// TwinCAT 3 PLC project CL_TelegramTxtLogLibrary
// Title: CL_TelegramTxtLogLibrary
// Company: CleanGreens SA
// Author: Massimo Lucano
// ProjectVersion: 2.2
// Description: Telegram API implementation, TextLOg implementation, Link between CL_DefectManager and Telegram and TextLog
// ProgramVersion: 3.1.4024.0
// libraries:
//   CL_DefectManager, * (CleanGreens SA)
//   CL_ErrorsDatabase, * (CleanGreens SA)
//   CL_CleanGreensObjectsLibrary, * (CleanGreens SA)
//   Tc2_Standard, * (Beckhoff Automation GmbH)
//   Tc2_System, * (Beckhoff Automation GmbH)
//   Tc2_Utilities, * (Beckhoff Automation GmbH)
//   Tc3_IotBase, * (Beckhoff Automation GmbH)
//   Tc3_IotCommunicator, * (Beckhoff Automation GmbH)
//   Tc3_JsonXml, * (Beckhoff Automation GmbH)
//   Tc3_Module, * (Beckhoff Automation GmbH)
// project tree:
//   DUTs/ enBOT_API.TcTLEO, E_MsgType.TcDUT, ST_getMe.TcDUT, ST_TelegramInit.TcDUT
//   / PlcTask.TcTTO
//   POUs/ CL_LinkDefectMgrToTelegramAndLog.TcPOU, CL_TelegramBOT.TcPOU, CL_TextLog.TcPOU
// real-time tasks:
//   TASK PlcTask: cycle T#10ms, priority 20, ADS port 350

CONFIGURATION CL_TelegramTxtLogLibrary
    RESOURCE PLC ON TwinCAT3
        TASK PlcTask(INTERVAL := T#10ms, PRIORITY := 20);
        PROGRAM Main WITH PlcTask : Main;
    END_RESOURCE
END_CONFIGURATION

// ---- DUTs/enBOT_API.TcTLEO
TYPE enBOT_API :
(
	none := 0, getMe := 1, sendMsg := 2, getUpdates := 3
);
END_TYPE

// ---- DUTs/E_MsgType.TcDUT
{attribute 'qualified_only'}
{attribute 'strict'}
TYPE E_MsgType :
(
	Alarm := 0,
  Info,
  Register
);
END_TYPE

// ---- DUTs/ST_getMe.TcDUT
TYPE ST_getMe :
STRUCT
	id 						              : ULINT;
	first_name				          : T_MaxString;//BOT name
	username				            : T_MaxString;//owner name
  is_bot					            : BOOL;
	can_join_groups			        : BOOL;
	can_read_all_group_messages : BOOL;
	supports_inline_queries	    : BOOL;
END_STRUCT
END_TYPE

// ---- DUTs/ST_TelegramInit.TcDUT
TYPE ST_TelegramInit :
STRUCT
  sBOTKey   		  : STRING(64);//BOT key to exchange operator messages
	sDebugID   		  : STRING(32);//chat group ID to send debug messages Info et Verbose
	sAlarmID   		  : STRING(32);//chat group ID to send Critical,Error,Warning alarms
	sBOTname  		  : STRING(40);
	sBOTusername  	: STRING(40);
END_STRUCT
END_TYPE

// ---- POUs/CL_LinkDefectMgrToTelegramAndLog.TcPOU
{attribute 'enable_dynamic_creation'}
FUNCTION_BLOCK CL_LinkDefectMgrToTelegramAndLog EXTENDS CL_MasterRootClass
VAR
  bInit                   : BOOL := FALSE;
	_DefectMngr             : REFERENCE TO CL_DefectManager;
  _TelegramBOT            : REFERENCE TO CL_TelegramBOT;
  _TxtLog                 : REFERENCE TO CL_TextLog;
  _ActTime                :	REFERENCE TO CL_ActTimeDate;
  
  indListAll 					    : UINT := 1;
  indListAct  				    : UINT := 1;

  _stConfigMsgBuild       : ST_ConfigMsgBuild;
  _stShow                 : ST_ShowMsgFields;
  
  _bShowRegisterMsg       : BOOL := FALSE;
  _bAllDefectsRegistered  : BOOL := FALSE;
	
	sTelegramMsg_P	        : POINTER TO T_StringBuffer;//used to generate very long Telegram messages limited to 3500 chars
	sTextOut_P              : POINTER TO T_StringBuffer;//used to generate short ADS console messages limited to 255 chars
  
	pDf			      		      : POINTER TO CL_Defect;
	iDf		        		      : ITF_Defect;
END_VAR

IF bInit THEN
  this^.Run(); 
END_IF

METHOD PRIVATE AddDateTime
VAR_IN_OUT
	sMsgTimeCreation	: T_MaxString;
END_VAR
VAR
  sDatetime         : T_MaxString;
END_VAR
(*
sBOTMsgTimeCreation^ := DT_TO_STRING(_objActTime_R.GetDateTime);
sBOTMsgTimeCreation^ := REPLACE(sBOTMsgTimeCreation^,' ',1,3);
sBOTMsgTimeCreation^ := CONCAT(' ',sBOTMsgTimeCreation^);
//sBOTMsgTimeCreation^ := CONCAT(sBOTMsgTimeCreation^,'%0A');
sBOTMsgTimeCreation^ := CONCAT(sBOTMsgTimeCreation^,'  ');
*)

(*
sMsgTimeCreation := concat(sMsgTimeCreation,_ActTime.GetStrDateTime());//2024-10-15-23:16:25
sMsgTimeCreation := REPLACE(sMsgTimeCreation,' ',1,11);
sMsgTimeCreation := CONCAT('Date: ', sMsgTimeCreation);
sMsgTimeCreation := CONCAT(sMsgTimeCreation,'  ');
*)

sMsgTimeCreation := CONCAT(sMsgTimeCreation,'  Date: ');
sDatetime := _ActTime.GetStrDateTime();//2024-10-15-23:16:25
sDatetime := REPLACE(sDatetime,' ',1,11);
sMsgTimeCreation := CONCAT(sMsgTimeCreation,sDatetime);
END_METHOD

PROPERTY PUBLIC AllDefectsRegistered : BOOL
GET
AllDefectsRegistered := _bAllDefectsRegistered;
END_GET
SET
_bAllDefectsRegistered := AllDefectsRegistered;
END_SET
END_PROPERTY

METHOD PRIVATE BuildMsg : BOOL
VAR_INPUT
  MsgType       : E_MsgType;
END_VAR
VAR
  sStartMsg     : T_MAXSTRING;
  
END_VAR
//%0A telegram new line
CASE MsgType OF
  E_MsgType.Alarm:
    sStartMsg := _stConfigMsgBuild.AlarmMsg.sStartMsg;
    _stShow := _stConfigMsgBuild.AlarmMsg;
  E_MsgType.Info:
    sStartMsg := _stConfigMsgBuild.InfoMsg.sStartMsg;
    _stShow := _stConfigMsgBuild.InfoMsg;
  E_MsgType.Register:
    sStartMsg := _stConfigMsgBuild.RegisterMsg.sStartMsg;
    _stShow := _stConfigMsgBuild.RegisterMsg;
END_CASE   
sTelegramMsg_P^ := '';
sTextOut_P^ := '';

BuildMsg := pDf^.BuildStringMsg(sMsgOut_P := sTelegramMsg_P, sTextOut_P := sTextOut_P, stShow := _stShow);
                                      
IF _stShow.bDateTime THEN 
  AddDateTime(sStartMsg);
END_IF  

IF _stShow.bTelegram THEN
  CONCAT2(ADR(sStartMsg),sTelegramMsg_P,sTelegramMsg_P,SIZEOF(sTelegramMsg_P^));
END_IF

IF _stShow.bTxtLog THEN
  CONCAT2(ADR(sStartMsg),sTextOut_P,sTextOut_P,SIZEOF(sTextOut_P^));
END_IF
END_METHOD

METHOD PUBLIC Init : BOOL
VAR_INPUT
  stIrrLine        : ST_LineReference;
  DefectMngr       : REFERENCE TO CL_DefectManager;
  TelegramBOT      : REFERENCE TO CL_TelegramBOT;
  TxtLog           : REFERENCE TO CL_TextLog;
  ActTime          : REFERENCE TO CL_ActTimeDate;
  stConfigMsg      : ST_ConfigMsgBuild;
END_VAR
VAR
  bufferSize       : UDINT;
END_VAR
bInit := Init := FALSE;
IF __ISVALIDREF(DefectMngr) AND __ISVALIDREF(TelegramBOT) AND __ISVALIDREF(TxtLog) and __IsValidRef(ActTime) THEN 
	_DefectMngr REF= DefectMngr;
  _TelegramBOT REF= TelegramBOT;
  _TxtLog REF= TxtLog;
  _ActTime REF= ActTime;
  
  MRCLineRef := stIrrLine;

  indListAll := indListAct := 1;

	_stConfigMsgBuild := stConfigMsg;
  _bShowRegisterMsg := _stConfigMsgBuild.bShowRegisterMsg;
  
  bufferSize := SIZEOF(T_StringBuffer)+4;
  sTelegramMsg_P := __NEW(BYTE, bufferSize);
  sTextOut_P := __NEW(BYTE, bufferSize);

  bInit := Init := sTelegramMsg_P <> 0 AND sTextOut_P <> 0;
END_IF
END_METHOD

PROPERTY PUBLIC RegisterAllMsgSent : BOOL
GET
RegisterAllMsgSent := not _bShowRegisterMsg;
END_GET
END_PROPERTY

METHOD PUBLIC Release : BOOL
bInit := FALSE;
IF sTelegramMsg_P <> 0  THEN 
  __DELETE(sTelegramMsg_P);
END_IF

IF sTextOut_P <> 0  THEN 
  __DELETE(sTelegramMsg_P);
END_IF

Release := sTelegramMsg_P = 0 AND sTextOut_P = 0;
END_METHOD

METHOD PRIVATE Run
VAR
  bDefectToSend	: BOOL;
END_VAR
IF NOT _TelegramBOT.IsBusy AND NOT _TxtLog.IsBusy THEN  
  
  IF _bShowRegisterMsg  THEN
    pDf := _DefectMngr.ListAll(indListAll,0);
    IF pDf <> 0 THEN
      iDf := pDf^;
      IF __QUERYPOINTER(iDf, pDf) THEN // Ctrl if address has the good interface (ITF_Default)
        RunRegister();
      END_IF//__QUERYPOINTER
    END_IF//_DefectMngr.List(indDfList,0) <> 0 
    //Telegram and TextLog not Busy --> increment at each cycle the Defect index
    indListAll := indListAll + 1;
    IF (indListAll > _DefectMngr.nMaxDefects) THEN //all Defect Register Messages sent
      indListAll := 1;
      //after first pass all register messages are sent, do not send anymore
      //the object can send starting from now Alarm and Info messages
      _bShowRegisterMsg := FALSE;
    END_IF 
  END_IF//_bShowRegisterMsg
  
  IF NOT _bShowRegisterMsg  THEN
    pDf := _DefectMngr.ListCurrent(indListAct);
    IF pDf <> 0 THEN
      iDf := pDf^;
      IF __QUERYPOINTER(iDf, pDf) THEN // Ctrl if address has the good interface (ITF_Default)
        IF pDf^.DefectToSend THEN 
          RunAlarm();
          RunInfo();
        END_IF
      END_IF//__QUERYPOINTER
    END_IF//_DefectMngr.ListCurrent(indDfList,0) <> 0 
    indListAct := indListAct + 1;
    IF (indListAct > _DefectMngr.nMaxDefectsView) THEN
      indListAct := 1;
    END_IF 
  END_IF//not _bShowRegisterMsg
ELSE
  //ADSLOGSTR(ADSLOG_MSGTYPE_LOG, 'Telegram busy','');//only for debug
  IF _TelegramBOT.IsError THEN 
    ADSLOGSTR(ADSLOG_MSGTYPE_LOG, 'Telegram error: Telegram server answer with HTTP error','');
  END_IF
END_IF//TelegramBOT and TextLog both are not busy
END_METHOD

METHOD PRIVATE Run_old
VAR
  bDefectToSend	: BOOL;
END_VAR
(*
IF NOT _TelegramBOT.IsBusy AND NOT _TxtLog.IsBusy THEN  
  
	IF _DefectMngr.List(indDfList,0) <> 0 THEN
		iDf := _DefectMngr.List(indDfList,0)^;
		IF __QUERYPOINTER(iDf, pDf) THEN // Ctrl if address has the good interface (ITF_Default)
      pDf := _DefectMngr.List(indDfList,0);  
      IF _bShowRegisterMsg then
        RunRegister();
        IF (indDfList > _DefectMngr.nMaxDefects) THEN //all Defect Register Messages sent
          _bShowRegisterMsg := false;//Register all defects done; the object can send starting from now Alarm and Info messages
				END_IF
			ELSE
        //condition OR pDf^.State = E_DefectState.OffAndNotAck added MPL date 16-11-2024
        bDefectToSend := pDf^.State = E_DefectState.Active OR pDf^.State = E_DefectState.ActiveAndAck OR pDf^.State = E_DefectState.OffAndNotAck;
        IF bDefectToSend THEN 
          RunAlarm();        
          RunInfo();
        END_IF
      END_IF
    END_IF//__QUERYPOINTER
  END_IF//_DefectMngr.List(indDfList,0) <> 0 

  //Telegram and TextLog not Busy --> increment at each cycle the Defect index
  indDfList := indDfList + 1;
  IF (indDfList > _DefectMngr.nMaxDefects) THEN	// Constant not accessible defect manager, or yes. Actually yes, but access through GVL not suitable!	
    indDfList := 1;
    _bShowRegisterMsg := false;//after first pass all register messages are sent, do not send anymore
  END_IF 
END_IF//TelegramBOT and TextLog both are not busy
*)
END_METHOD

METHOD PRIVATE RunAlarm
VAR_INPUT
END_VAR
//TcEventSeverity : (Verbose:=0, Info:=1, Warning:=2, Error:=3, Critical:=4);
IF pDf^.CanSendAlarmMsg AND (pDf^.Severity > TcEventSeverity.Info) THEN //Telegram msg not yet sent   
  //Critical, Error and Warning Defect are sent to Alarm group
  IF BuildMsg(E_MsgType.Alarm) THEN
    IF _stShow.bTxtLog THEN 
      _TxtLog.RequWriteMsg(sTextOut_P);
    END_IF
    IF _stShow.bTelegram THEN
      _TelegramBOT.RequSendMsgToAlarm(sTelegramMsg_P);
    END_IF
  END_IF					
END_IF//pDf^.Severity... and pDf^.CanSendTelegramAlarmMsg
END_METHOD

METHOD PRIVATE RunInfo
VAR_INPUT
END_VAR
//TcEventSeverity : (Verbose:=0, Info:=1, Warning:=2, Error:=3, Critical:=4);
//sendMsgToAlarm and sendMsgToInfo cannot be executed together; sendMsgToInfo can be requested only once AlarmMsgAlreadySent is true and TelegramBOT is again not busy
//IF (pDf^.CanSendInfoMsg AND (pDf^.Severity <= TcEventSeverity.Info)) OR (pDf^.CanSendInfoMsg AND (pDf^.Severity > TcEventSeverity.Info) AND pDf^.AlarmMsgAlreadySent) THEN
IF (pDf^.CanSendInfoMsg AND (pDf^.Severity <= TcEventSeverity.Info)) THEN
  //Verbose and Info Defect are sent only to InfoDebug group
  IF BuildMsg(E_MsgType.Info) THEN
    IF _stShow.bTelegram THEN
      _TelegramBOT.RequSendMsgToInfo(sTelegramMsg_P);
    END_IF
    IF _stShow.bTxtLog THEN 
      _TxtLog.RequWriteMsg(sTextOut_P);
    END_IF
  END_IF
END_IF//pDf^.Severity... and pDf^.CanSendTelegramAlarmMsg
END_METHOD

METHOD PRIVATE RunRegister
IF pDf^.CanSendRegisterMsg AND _bShowRegisterMsg THEN //all Defect registered are sent
  IF BuildMsg(E_MsgType.Register) THEN
   IF _stShow.bTxtLog THEN 
    _TxtLog.RequWriteMsg(sTextOut_P);
   END_IF
   IF _stShow.bTelegram THEN
    _TelegramBOT.RequSendMsgToInfo(sTelegramMsg_P);
   END_IF
  END_IF
END_IF
END_METHOD

METHOD PRIVATE TelegramMsgFilter : BOOL
VAR_INPUT
	sDatabaseMsg	:	T_MaxString;
END_VAR
VAR_OUTPUT
	sTelegramMsg	:	T_MaxString;
END_VAR
VAR
	sTelegramTmp	:	T_MaxString;
	i:	INT;
	iSafe:	INT;
	iLengthStr:	INT	:= 0;
	iNonAsciiPos:	INT;
	iNumAsciiChar:	UDINT;

END_VAR

VAR CONSTANT
		// Language tables - hardcoded here since part of the algorithm, and meaningless to keep them outside.
	sASCIIcompatCharFR_AR : ARRAY [1..2,1..28] OF STRING := ['à','â','é','è','ê','ë','î','ï','ô','ù','û','ü','ÿ','ç',
																															'À','Â','É','È','Ê','Ë','Î','Ï','Ô','Ù','Û','Ü','Ÿ','Ç',
																															2('a'),4('e'),2('i'),'o',3('u'),'y','c',
																															2('A'),4('E'),2('I'),'O',3('U'),'Y','C'];
	sASCIIcompatCharDE_AR :	ARRAY [1..2,1..7] OF STRING  := ['Ä','ä','Ö','ö','Ü','ü','ß',
																															'Ae','ae','Oe','oe','Ue','ue','ss'];
END_VAR

sTelegramTmp := sDatabaseMsg;
IF NOT F_StringIsASCII(pSTRING := ADR(sTelegramTmp), nLen => iNumAsciiChar) THEN
	iLengthStr := LEN(sTelegramTmp);
//	IF C.sLangErrors = 'fr' THEN
	IF  _DefectMngr.ErrorDB.sMsgLang = 'fr' THEN
			FOR i:=1 TO 28 BY 1 DO
				iSafe := 0;
				REPEAT
					iNonAsciiPos := FIND(sTelegramTmp,sASCIIcompatCharFR_AR[1,i]);	// Table to store inside the object, as never used elsewhere and fixed sized.
					IF iNonAsciiPos <> 0 THEN
						sTelegramTmp := REPLACE(sTelegramTmp,sASCIIcompatCharFR_AR[2,i],1,iNonAsciiPos);
					END_IF
					iSafe := iSafe + 1;
				UNTIL iNonAsciiPos = 0 OR iSafe > iLengthStr
				END_REPEAT;	
			END_FOR
//	ELSIF C.sLangErrors = 'de' THEN
	ELSIF  _DefectMngr.ErrorDB.sMsgLang = 'de' THEN
		FOR i:=1 TO 7 BY 1 DO
		iSafe := 0;
			REPEAT
				FIND(sTelegramTmp,sASCIIcompatCharDE_AR[1,i]);
				IF iNonAsciiPos <> 0 THEN
					REPLACE(sTelegramTmp,sASCIIcompatCharDE_AR[2,i],1,iNonAsciiPos); // Caution, the length of the string is increasing
				END_IF
			iSafe := iSafe + 1;
			UNTIL iNonAsciiPos = 0 OR iSafe > 2*iLengthStr
			END_REPEAT
		END_FOR
	END_IF
END_IF
sTelegramMsg := sTelegramTmp;

//only to reproduce the bug without filtering
//sTelegramMsg := sDatabaseMsg;
END_METHOD

END_FUNCTION_BLOCK

// ---- POUs/CL_TelegramBOT.TcPOU
{attribute 'enable_dynamic_creation'}
FUNCTION_BLOCK CL_TelegramBOT EXTENDS CL_MasterRootClass
VAR CONSTANT //constant configuration parameters fro FB_IotHttpClient configuration
	sHostNameC 					: T_MaxString:='api.telegram.org';
	nHostPortC  				: UINT := 443; //https port
	bKeepAliveC 				: BOOL := FALSE;
	bNoServerCertCheckC : BOOL := TRUE;
	tConnectionTimeoutC : TIME := T#10S;
END_VAR
VAR
	boBOT_MSGOk 				: BOOL := FALSE;
		
	sBOTKey 						: T_MaxString;// BOT key to exchange operator messages
	sDebugID 						: STRING(64);//32
	sAlarmID 						: STRING(64);//32
	sBOTname 						: STRING(64);//40
	sBOTusername 				: STRING(64);//40
	
	bInit		            : BOOL := FALSE;
 	
	fbHttpClientTelegram: FB_IotHttpClient;//HTTP client communication
	fbBOTRequest   			: FB_IotHttpRequest;
	
	sBOTMsgBuffer_P			: POINTER TO T_StringBuffer;//STRING(2000);//string buffer
	sBOT_APIMethod_P 		: POINTER TO T_StringBuffer;//STRING(3500);//used in HTTPGetTelegram
	sBOTReturnContent_P : POINTER TO T_StringBuffer;//STRING(2000);//used in HTTPGetTelegram
  
	RisingEdge          : R_TRIG;
	HTTPGetTelegramStm  : BYTE := 0;
  nBOTReqCnt          : UDINT := 0;    
  nBOTContentCnt      : UDINT := 0;
    
  nErrCount           : UDINT;
	bBOTSend						: BOOL;
	bBOTHTTPError			  : BOOL := FALSE;
	bBOTBusy            : BOOL := FALSE; 
	
	//used in
	bJSONReturnExec			: BOOL := FALSE;
	JSONReturnStm				: enBOT_API := enBOT_API.none;
	nJSONResCnt         : UDINT := 0;
	
	//returned values from getMe
	stJsonGetMe					: ST_getMe;
	bJsonGetMe					: BOOL;
	bBOTCorret					: BOOL  := TRUE; //the BOT is correctly identified after the initial getMe Api call 
END_VAR
{attribute 'TcEncoding':='UTF-8'}

//IMPORTANT ATTENTION: forbidden words for Telegram messages otherwise FB_IotHttpRequest FAILS!! Forbidden words: HandlingLine HMI
IF bInit THEN
	IF fbHttpClientTelegram.bConfigured AND bBOTCorret THEN
		fbHttpClientTelegram.Execute();
		HTTPGetTelegramExec();
		JSONBOTReturnExec();
	END_IF
END_IF

METHOD PRIVATE HTTPGetTelegramExec
VAR
   nBOTReturnContentSize 		: UDINT;
	 HTTPStatusCodeFromServer	: UINT;
END_VAR
IF (bBOTSend) THEN
	RisingEdge(CLK:= TRUE );
	CASE HTTPGetTelegramStm OF
		0: IF RisingEdge.Q THEN 
				IF fbBOTRequest.SendRequest(sUri:=sBOT_APIMethod_P^, fbClient:=fbHttpClientTelegram, eRequestType:=ETcIotHttpRequestType.HTTP_Get, 0, 0, 0) THEN                
					HTTPGetTelegramStm:= 1;
					nBOTReqCnt:= nBOTReqCnt+1;
					bBOTBusy:= TRUE;
					bBOTHTTPError:= FALSE;
				END_IF                    
    	END_IF
		1: IF NOT fbBOTRequest.bBusy THEN
        bBOTHTTPError:= TRUE;
        IF NOT fbBOTRequest.bError THEN  
          bBOTHTTPError:= NOT fbBOTRequest.GetContent(pContent:= sBOTReturnContent_P,
					nContentSize:= nBOTReturnContentSize:= SIZEOF(T_StringBuffer),
					bSetNullTermination:= TRUE);
					IF JSONReturnStm = enBOT_API.getUpdates THEN
						bBOTHTTPError := FALSE;
						//the JSON answer from getUpdates methos could be very large; in this case a truncated answer will be stored in sBOTReturnContent
						//fbBOTRequest.GetContent will return an error -> in this case the error is always cleared
					END_IF
					bBOTSend := FALSE; //do not execute any longer HTTPGetTelegramExec
					//bBOTError:= FALSE -> ok sBOTReturnContent returned good value
					HTTPStatusCodeFromServer := fbBOTRequest.nStatusCode;
					IF NOT bBOTHTTPError AND HTTPStatusCodeFromServer >= 200 AND HTTPStatusCodeFromServer < 300 THEN
						bJSONReturnExec := TRUE;
						nBOTContentCnt:= nBOTContentCnt+1;
					ELSE
						bBOTHTTPError := TRUE;//server answer with HTTP error
            //ADSLOGSTR(ADSLOG_MSGTYPE_LOG, 'Telegram error: Telegram server answer with HTTP error','');//only debug
					END_IF
        END_IF
				RisingEdge(CLK:= FALSE);
				HTTPGetTelegramStm := 0;
				bBOTBusy:= FALSE;
				IF bBOTHTTPError THEN
					nErrCount:= nErrCount+1;
				END_IF
    	END_IF
	END_CASE
END_IF
END_METHOD

METHOD PUBLIC Init : BOOL
VAR_INPUT
  stIrrLine       : ST_LineReference;
	stTelegramIn    : ST_TelegramInit;
END_VAR

VAR	
	fbFormatStr			: FB_FormatString;
	sHTTP_BOTAnswer	: STRING(500);
  bufferSize      : UDINT;
END_VAR
bInit := Init := LEN(stTelegramIn.sBOTKey) >0 AND LEN(stTelegramIn.sBOTusername) >0 AND LEN(stTelegramIn.sBOTname) >0 AND (LEN(stTelegramIn.sDebugID) >0 OR Len(stTelegramIn.sAlarmID) > 0);
IF Init THEN	
  MRCLineRef := stIrrLine;
  
  sBOTKey := stTelegramIn.sBOTKey;
  sDebugID := stTelegramIn.sDebugID;
  sAlarmID := stTelegramIn.sAlarmID;
  sBOTname := stTelegramIn.sBOTname;
  sBOTusername := stTelegramIn.sBOTusername;
  
  bufferSize := SIZEOF(T_StringBuffer)+4;
  sBOTMsgBuffer_P := __NEW(BYTE, bufferSize);
  sBOT_APIMethod_P := __NEW(BYTE, bufferSize);
  sBOTReturnContent_P := __NEW(BYTE, bufferSize);
  
  bInit := Init := sBOTMsgBuffer_P <> 0 AND sBOT_APIMethod_P <> 0 AND sBOTReturnContent_P <> 0;
  IF Init THEN
    sBOTMsgBuffer_P^:= '';
    sBOT_APIMethod_P^:= '';
    sBOTReturnContent_P^:= '';
    IF NOT fbHttpClientTelegram.bConfigured THEN
      //fbHttpClientTelegram.stTLS.sCA:='C:\TwinCAT\3.1\Config\Certificates\TelegramRoot.cer';  //server certificate
      fbHttpClientTelegram.sHostName := sHostNameC;
      fbHttpClientTelegram.nHostPort := nHostPortC;
      fbHttpClientTelegram.bKeepAlive := bKeepAliveC;
      fbHttpClientTelegram.tConnectionTimeout:=tConnectionTimeoutC;
      fbHttpClientTelegram.stTLS.bNoServerCertCheck:=bNoServerCertCheckC; //avoid certificate
      fbHttpClientTelegram.Execute();		
      bInit := Init := TRUE;
      bBOTBusy := FALSE;//no request
      RequGetMe(); //must be called after having initialized bInit //getUpdates(); 
      bBOTBusy := TRUE; //must be set to TRUE -> HTTP BOT Api request getME still not executed and done
    ELSE
      bInit := Init := FALSE;
    END_IF
  END_IF
END_IF
END_METHOD

PROPERTY PUBLIC IsBusy : BOOL
GET
IF bInit THEN
  IsBusy := bBOTBusy;
ELSE
  IsBusy := TRUE;
END_IF
END_GET
END_PROPERTY

PROPERTY PUBLIC IsError : BOOL
GET
IF bInit THEN
  IsError := bBOTHttpError;
ELSE
  IsError := true;
END_IF
END_GET
END_PROPERTY

METHOD PRIVATE JSONBOTReturnExec
VAR
	bJSONOk: BOOL;
END_VAR
IF bJSONReturnExec THEN
	CASE JSONReturnStm OF
		enBOT_API.none: 
			bJSONReturnExec := FALSE;
			
		enBOT_API.getMe:
			bJSONOk := JSONParser_getMe();
			bJSONReturnExec := FALSE; //stop execution 
			JSONReturnStm := enBOT_API.none;
			
		enBOT_Api.sendMsg:
			//bJSONOk := JSONParser_sendMsg();  TO DO
			bJSONReturnExec := FALSE; //stop execution 
			JSONReturnStm := enBOT_API.none;
		
		enBOT_API.getUpdates:
			//bJSONOk := JSONParser_getUpdates();  To DO
			bJSONReturnExec := FALSE; //stop execution 
			JSONReturnStm := enBOT_API.none;			
	END_CASE
	sBOTReturnContent_P^ := '';
END_IF
END_METHOD

METHOD PRIVATE JSONParser_getMe : BOOL
VAR
	jsonDoc 	: SJsonValue;
	fbJson  	: FB_JsonDomParser;

	jsonPtmp, jsonP_result	: SJsonValue;
	jsonS_ok, jsonS_result	: T_MaxString;
	
  	fbJsonDataType  : FB_JsonReadWriteDataType;
END_VAR
JSONParser_getMe := FALSE;
jsonDoc := fbBOTRequest.GetJsonDomContent(fbJson);
IF jsonDoc <> 0 THEN
	jsonDoc := fbJson.ParseDocument(sBOTReturnContent_P^);
	IF jsonDoc <> 0 THEN
		jsonPtmp := fbJson.FindMember(jsonDoc, 'ok');
		jsonP_result := fbJson.FindMember(jsonDoc, 'result');
		IF (jsonPtmp <> 0) AND (jsonP_result <> 0) THEN
			jsonS_ok := fbJson.GetJson(jsonPtmp);
			bJsonGetMe := StrEqual(jsonS_ok, 'true');
			IF bJsonGetMe THEN
				jsonS_result := fbJson.GetJson(jsonP_result);
				IF jsonS_result <> '' THEN 
					//the following line is not correctly executed in library !!!   why?
					//JSONParser_getMe := fbJsonDataType.SetSymbolFromJson(jsonS_result,'ST_getMe',SIZEOF(stJsonGetMe), ADR(stJsonGetMe));
					//must be replaced with the following lines!!!!!
					jsonPtmp := fbJson.FindMember(jsonP_result, 'is_bot');				
					stJsonGetMe.is_bot := StrEqual(fbJson.GetJson(jsonPtmp), 'true');
					jsonPtmp := fbJson.FindMember(jsonP_result, 'first_name');
					stJsonGetMe.first_name := fbJson.GetJson(jsonPtmp);
					stJsonGetMe.first_name := DELETE(stJsonGetMe.first_name,1,1);
					stJsonGetMe.first_name := DELETE(stJsonGetMe.first_name,1,len(stJsonGetMe.first_name));
					jsonPtmp := fbJson.FindMember(jsonP_result, 'username');
					stJsonGetMe.username := fbJson.GetJson(jsonPtmp,);
					stJsonGetMe.username := DELETE(stJsonGetMe.username,1,1);
					stJsonGetMe.username := DELETE(stJsonGetMe.username,1,len(stJsonGetMe.username));					
					nJSONResCnt:= nJSONResCnt+1;
					JSONParser_getMe := TRUE;
				END_IF
			END_IF
		END_IF
	END_IF   
END_IF

bBOTCorret := JSONParser_getMe AND stJsonGetMe.is_bot AND StrEqual(stJsonGetMe.first_name, sBOTname) AND StrEqual(stJsonGetMe.username, sBOTusername);
END_METHOD

METHOD PUBLIC Release : BOOL
bInit := FALSE;
IF sBOTMsgBuffer_P <> 0  THEN 
  __DELETE(sBOTMsgBuffer_P);
END_IF

IF sBOT_APIMethod_P <> 0 THEN 
  __DELETE(sBOT_APIMethod_P);
END_IF

IF sBOTReturnContent_P <> 0 THEN 
  __DELETE(sBOTReturnContent_P);
END_IF

Release := sBOTMsgBuffer_P = 0 AND sBOT_APIMethod_P = 0 AND sBOTReturnContent_P = 0;
END_METHOD

METHOD PUBLIC RequGetMe
VAR
	fbFormatStr	  : FB_FormatString;
	bTmp		      : BOOL;
END_VAR
IF fbHttpClientTelegram.bConfigured AND NOT IsBusy AND bInit THEN //NOT bBOTBusy -> the BOT Api command can be executed
  fbFormatStr(
		sFormat	:= '/bot%s/getMe', //BOT Api method getMe
		arg1	:= F_STRING(sBOTKey), 
		bError	=> bTmp,  
		nErrId	=> , 
		sOut	=> sBOT_ApiMethod_P^);//write Telegram BOT API HTTP string
		
		bBOTSend := NOT bTmp; //enable HTTPGetTelegram method execution  
		IF NOT bTmp THEN
			JSONReturnStm := enBOT_API.getMe; //JSON parser is instructed to parse a return msg from getMe BOT Api
		ELSE
			sBOT_ApiMethod_P^:='';  //clear Telegram BOT API HTTP string
			JSONReturnStm := enBOT_API.none; //JSON parser do nothing
		END_IF
END_IF
END_METHOD

METHOD PUBLIC RequGetUpdates
VAR
	fbFormatStr	  : FB_FormatString;
	bTmp		      : BOOL;
END_VAR
IF fbHttpClientTelegram.bConfigured AND NOT IsBusy AND bInit THEN  //NOT bBOTBusy -> the BOT Api command can be executed
	fbFormatStr(
		sFormat	:= '/bot%s/getUpdates', //BOT Api method getMe
		arg1	:= F_STRING(sBOTKey), 
		bError	=> bTmp,  
		nErrId	=> , 
		sOut	=> sBOT_ApiMethod_P^);//write Telegram BOT API HTTP string
		
		bBOTSend := NOT bTmp; //enable HTTPGetTelegram method execution  
		IF NOT bTmp THEN
			JSONReturnStm := enBOT_API.getUpdates; //JSON parser is instructed to parse a return msg from getUpdates BOT Api
		ELSE
			sBOT_ApiMethod_P^:='';  //clear Telegram BOT API HTTP string
			JSONReturnStm := enBOT_API.none; //JSON parser do nothing
		END_IF
END_IF
END_METHOD

METHOD PUBLIC RequSendMsgToAlarm
VAR_INPUT
	sTxtIn				: POINTER TO T_StringBuffer;
END_VAR
VAR
	fbFormatStr		: FB_FormatString;
	bTmpErr				: BOOL;
	len 					: UINT;
  sTmp          : T_MaxString;
END_VAR
IF fbHttpClientTelegram.bConfigured AND NOT IsBusy AND bInit THEN //NOT bBOTBusy -> the BOT Api command can be executed
  //ATTENTION DON'T WRITE INSIDE THE POINTER sTxtIn!!!
  sBOTMsgBuffer_P^:='';//cleare previous stored data
  len := SIZEOF(T_StringBuffer);
  CONCAT2(sBOTMsgBuffer_P, sTxtIn, sBOTMsgBuffer_P, len);
	//Telegram API new line character is %0A
	//to insert it inside format string the Telegram use %%0A
  sTmp := sAlarmID;
	fbFormatStr(
		sFormat	:= '/bot%s/sendMessage?chat_id=%s&text=', 
		arg1	:= F_STRING(sBOTKey), 
		arg2	:= F_STRING(sTmp), 
		bError	=> bTmpErr,  
		nErrId	=> , 
		sOut	=> sBOT_ApiMethod_P^);
		
		//CONCAT2 handles long string; fbFormatStr fails with long string
		IF NOT bTmpErr THEN
			len := SIZEOF(T_StringBuffer);
			bTmpErr := NOT CONCAT2(sBOT_ApiMethod_P,sBOTMsgBuffer_P,sBOT_ApiMethod_P, len);//write Telegram BOT API HTTP string
			JSONReturnStm := enBOT_API.sendMsg; //JSON parser is instructed to parse a return msg from sed message BOT Api
		END_IF
		bBOTSend := NOT bTmpErr; //enable HTTPGetTelegram method execution,  	
		IF bTmpErr THEN
			sBOT_ApiMethod_P^:='';  //clear Telegram BOT API HTTP string
			JSONReturnStm := enBOT_API.none; //JSON parser do nothing
		END_IF
END_IF
END_METHOD

METHOD PUBLIC RequSendMsgToInfo
VAR_INPUT
	sTxtIn				: POINTER TO T_StringBuffer;
END_VAR
VAR
	fbFormatStr		: FB_FormatString;
	bTmpErr				: BOOL;
	len 					: UINT;
  sTmp          : T_MaxString;
END_VAR
IF fbHttpClientTelegram.bConfigured AND NOT IsBusy AND bInit THEN //NOT bBOTBusy -> the BOT Api command can be executed
  //ATTENTION DON'T WRITE INSIDE THE POINTER sTxtIn!!!
  sBOTMsgBuffer_P^:='';//cleare previous stored data
  len := SIZEOF(T_StringBuffer);
  CONCAT2(sBOTMsgBuffer_P, sTxtIn, sBOTMsgBuffer_P, len);

	//Telegram API new line character is %0A
	//to insert it inside la format string the Telegram use %%0A
  sTmp := sDebugID;
	fbFormatStr(
		sFormat	:= '/bot%s/sendMessage?chat_id=%s&text=', 
		arg1	:= F_STRING(sBOTKey), 
		arg2	:= F_STRING(sTmp), 
		bError	=> bTmpErr,  
		nErrId	=> , 
		sOut	=> sBOT_ApiMethod_P^);
		
		//CONCAT2 handles long string
		IF NOT bTmpErr THEN
			len := SIZEOF(T_StringBuffer);
			bTmpErr := NOT CONCAT2(sBOT_ApiMethod_P,sBOTMsgBuffer_P,sBOT_ApiMethod_P,len);//write Telegram BOT API HTTP string
			JSONReturnStm := enBOT_API.sendMsg; //JSON parser is instructed to parse a return msg from sed message BOT Api
		END_IF
		bBOTSend := NOT bTmpErr; //enable HTTPGetTelegram method execution  	
		IF bTmpErr THEN
			sBOT_ApiMethod_P^:='';  //clear Telegram BOT API HTTP string
			JSONReturnStm := enBOT_API.none; //JSON parser do nothing
		END_IF
END_IF
END_METHOD

METHOD PRIVATE StrEqual : BOOL
VAR_INPUT
	Str1 : T_MaxString;
	Str2 : T_MaxString;
END_VAR
StrEqual := (LEN(Str1) = LEN(Str2)) AND (FIND(Str1, Str2) = 1);
END_METHOD

END_FUNCTION_BLOCK

// ---- POUs/CL_TextLog.TcPOU
FUNCTION_BLOCK CL_TextLog EXTENDS CL_MasterRootClass
VAR
  bInit           : BOOL := FALSE;
	bBusy						: BOOL := FALSE;
  bRequWrite      : BOOL;
	bError					: BOOL;
	nErrId					: UDINT;  

	step						: DWORD 	:= 0;
  
  sBuffer				  : POINTER TO T_StringBuffer;//text to be written
  nByteToWrite    : UDINT;
  nByteWritten    : UDINT;

	sNetId					: T_AmsNetId := '';	(* TwinCAT system network address *)
  sFileName				: T_MaxString; (* CSV source file path and name *)
  hFile						: UINT		:= 0;(* File handle of the source file *)
	fbFileOpen			: FB_FileOpen;(* Opens file *)
	fbFileClose			: FB_FileClose;(* Closes file *)
	fbFileWrite			: FB_FileWrite;
END_VAR

IF bInit THEN
  THIS^.Run();
END_IF

METHOD Init : BOOL
VAR_INPUT
  stIrrLine     : ST_LineReference;
  sPathIn       : T_MaxString;
END_VAR
Init := bInit := FALSE;
IF sPathIn <> '' THEN 
	Init := bInit := TRUE;
	MRCLineRef := stIrrLine;
  sFileName := sPathIn;
  RequOpenTxtLog();
END_IF
END_METHOD

METHOD PRIVATE InitAllVars
bRequWrite	:= FALSE;
sNetId := '';	
hFile	:= 0;
bBusy 	:= FALSE;
bError	:= FALSE;
nErrId	:= 0;
sBuffer := 0;
step := 110;
END_METHOD

PROPERTY PUBLIC IsBusy : BOOL
GET
IF bInit THEN
  IsBusy := bBusy;
ELSE
  IsBusy := true;
END_IF
END_GET
END_PROPERTY

PROPERTY PUBLIC IsError : BOOL
GET
IF bInit THEN
  IsError := bError;
ELSE
  IsError := TRUE;
END_IF
END_GET
END_PROPERTY

METHOD PUBLIC Release : BOOL
VAR_INPUT
END_VAR
RequCloseTxtLog();//close text file
END_METHOD

METHOD PRIVATE RequCloseTxtLog
VAR_INPUT
END_VAR
IF NOT bBusy THEN
  bBusy := TRUE;
  step := 10;
END_IF
END_METHOD

METHOD PRIVATE RequOpenTxtLog
IF NOT bBusy THEN
  InitAllVars();
  step := 1;
  bBusy := TRUE;
END_IF
END_METHOD

METHOD PUBLIC RequWriteMsg
VAR_input
	sTxtIn				: POINTER TO T_StringBuffer;
END_VAR
IF NOT bBusy AND sTxtIn <> 0 THEN
  sBuffer := sTxtIn;
  bRequWrite := TRUE;
  step := 3;
ELSE
  bRequWrite := FALSE;
  step := 3;
END_IF
END_METHOD

METHOD PRIVATE Run
VAR
END_VAR
CASE step OF
  1://open text file
    fbFileOpen(  bExecute := FALSE  );
    fbFileOpen( sNetId := sNetId, sPathName := sFileName, nMode := FOPEN_MODEWRITE OR FOPEN_MODETEXT,(* Open file in TEXT mode! *)
                ePath := PATH_GENERIC, bExecute := TRUE );
    step := 2;

	2://Wait until open not busy 
		fbFileOpen( bExecute := FALSE, bError => bError, nErrID => nErrID, hFile => hFile );
		IF NOT fbFileOpen.bBusy THEN
			IF NOT fbFileOpen.bError THEN
        bBusy := FALSE;
				step := 3;
			ELSE(* Error: path not found or unable to create the file *)
				step := 100;
			END_IF
		END_IF

  3: //wait to execute a new write;
    IF bRequWrite AND NOT bBusy THEN 
      bRequWrite := FALSE;
      bBusy := TRUE;
      step := 4;
		END_IF
    
	4://start write data
    nByteToWrite := len2(sBuffer);
		fbFileWrite( bExecute := FALSE );
		fbFileWrite( sNetId := sNetId, hFile := hFile, pWriteBuff := sBuffer, cbWriteLen := nByteToWrite,  bExecute := TRUE );
		step := 5;

	5://Wait until write operation not busy 
		fbFileWrite( bExecute := FALSE, bError => bError, nErrID => nErrID, pWriteBuff := sBuffer, cbWrite => nByteWritten );
		IF NOT fbFileWrite.bBusy THEN
			IF NOT fbFileWrite.bError AND (nByteWritten = nByteToWrite) THEN
				step := 3;
        bBusy := FALSE;
			ELSE// Error
				step := 100;
			END_IF
		END_IF

	10://Close text file
		fbFileClose( bExecute := FALSE );
		fbFileClose( sNetId := sNetId, hFile := hFile, bExecute := TRUE );
		step := 11;

	11://Wait until close not busy
		fbFileClose( bExecute := FALSE, bError => bError, nErrID => nErrID );
		IF ( NOT fbFileClose.bBusy ) THEN
			hFile := 0;
			step := 100;
		END_IF

	100: //Error or ready step => cleanup
		IF ( hFile <> 0 ) THEN
			step := 10; //Close the source file
		ELSE
			bBusy := FALSE;
			step := 110;
		END_IF
  
  110:
    ;//do nothinh parked after calling Release or Error

END_CASE
END_METHOD

END_FUNCTION_BLOCK
